ABB RobotStudio station: TPL01.rspag

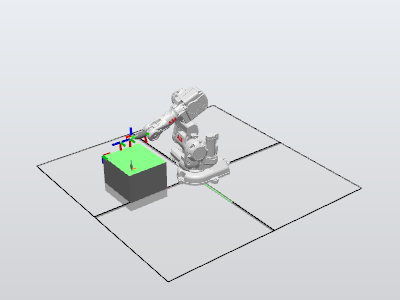
--- station ---
Station Project2 (saved by RobotStudio 25.5.11605.0)
Controller IRB140_6_81
  mechanical unit ROB_1: IRB140_6_81_C_03, 6 joints, base frame (0, 0, 0) mm
Layout (positions relative to the parent item):
  - IRB140_6_81_C_03 [mechanism, from %ABB.RobotStudio.Models.IRB140%\IRB140_6_81_C_G_03.rslib] at (0, 0, 0) mm; joint values [-0.1496, -0.0274, 0.4762, 2.8072, 0.4714, -2.4487] (rad or m)
  - Mesa [part], size 365 x 405 x 340 mm
  - Perno [part] at (730, 340, 177) mm, rotated rx 90 ry 0 rz -90 deg, size 20 x 100 x 20 mm
  - Pinza [mechanism] at (463, -60, 547) mm, rotated rx 90 ry 67.5 rz 90 deg
      TCP Pinza at (0, 0, 137) mm, rotated rx 0 ry 0 rz -22.5 deg
      links: Dummy
Attachment: Pinza is attached to IRB140_6_81_C_03 / Link6
Attachment: REF_Mesa is attached to Mesa
Attachment: REF_perno is attached to Perno
EventTableEntry 2314: ActivationMode=2, Cyclic=false, Group=, Trigger=DO_Pinza 2315, Actions=[EventTableActionAttach 2316], Comment=
EventTableTriggerIO 2315: Operator=0, IOValue=[1], IRC5Controller=? -1, SignalSource=IRB140_6_81 1261
EventTableActionAttach 2316: MountObject=false, FlangeIndext=0, FindNearest=false, AttachmentParent=Pinza 2308, AttachmentChild=Perno 2304, Offset=[X=1, Y=0, Z=0, W=0, X=0, Y=1, Z=0, W=0, X=0, Y=0, Z=1, W=0, X=0, Y=0, Z=0, W=1]
EventTableEntry 2317: ActivationMode=2, Cyclic=false, Group=, Trigger=DO_Pinza 2318, Actions=[EventTableActionDetach 2319], Comment=
EventTableTriggerIO 2318: Operator=0, IOValue=[0], IRC5Controller=? -1, SignalSource=IRB140_6_81 1261
EventTableActionDetach 2319: AttachmentParent=Pinza 2308, AttachmentChild=Perno 2304
Collision set CollisionSet_1: Perno against Mesa, near miss 0.005 m
EventTableTriggerIO 2517: Operator=0, IOValue=[1], IRC5Controller=? -1, SignalSource=IRB140_6_81 1261
EventTableTriggerIO 2518: Operator=0, IOValue=[0], IRC5Controller=? -1, SignalSource=IRB140_6_81 1261
Targets, tools, work objects and paths stored in the station and not in the controller backup, written as RAPID:
! task T_ROB1
MODULE Module1
  CONST robtarget home_10:=[[624.937,0,611],[1,0,0,0],[0,0,0,0],[9E+09,9E+09,9E+09,9E+09,9E+09,9E+09]];
ENDMODULE


--- Controller Data/IRB140_6_81/RAPID/TASK1/PROGMOD/CalibData.mod ---
MODULE CalibData
    PERS tooldata Pinza:=[TRUE,[[0,0,137],[0.98078528,0,0,-0.195090322]],[0.5,[0,0,100],[1,0,0,0],0,0,0]];
    TASK PERS wobjdata REF_Mesa:=[FALSE,TRUE,"",[[665,-400,260],[0,0,1,0]],[[0,0,0],[1,0,0,0]]];
    TASK PERS wobjdata REF_perno:=[FALSE,TRUE,"",[[400,180,130],[0.707106781,0.707106781,0,0]],[[0,0,0],[1,0,0,0]]];
ENDMODULE

--- Controller Data/IRB140_6_81/RAPID/TASK1/PROGMOD/Module1.mod ---
MODULE Module1
    CONST robtarget INSERTAR_PIEZA:=[[65,340,3],[1,0,0,0],[-1,1,-2,0],[9E+09,9E+09,9E+09,9E+09,9E+09,9E+09]];

    VAR robtarget TOMAR_PIEZA;
    !caso 1
    CONST robtarget TOMAR_PIEZA_VERTICAL:=[[0,0,10],[0.5,0.5,-0.5,0.5],[0,0,0,0],[9E+09,9E+09,9E+09,9E+09,9E+09,9E+09]];
    !caso 2
    CONST robtarget TOMAR_PIEZA_HORIZONTAL:=[[0,0,10],[1,0,0,0],[0,0,0,0],[9E+09,9E+09,9E+09,9E+09,9E+09,9E+09]];

    !Definicion de herramienta con perno
    PERS tooldata TCP_perno := [TRUE,[[83.1492,-34.4415,137],[0.69352,0.13795,0.69352,-0.13795]],[0.5,[0,0,100],[1,0,0,0],0,0,0]];

    !Transformacion pinza a perno
    VAR pose pinza_to_perno := [[90,0,0], [0,0,0,0]];

    VAR num MODO_PICK := 0; ! MODO_VERICAL = 0, MODO_HORIZONTAL = 1

    PROC main()

        init;
        test_path;

    ENDPROC

    PROC test_path()

        aproximar_perno;

        cerrar_pinza;

        aproximar_hueco;

        abrir_pinza;

        ir_inicio;

    ENDPROC


    PROC init()
        !Calculo de transformaciones de herramientas
        IF MODO_PICK = 0 THEN
            pinza_to_perno := [[90,0,0], OrientZYX(0,90,0)];
            TOMAR_PIEZA := TOMAR_PIEZA_VERTICAL;
        ELSE
            pinza_to_perno := [[0,0,90], OrientZYX(0,0,0)];
            TOMAR_PIEZA := TOMAR_PIEZA_HORIZONTAL;
        ENDIF

        TCP_perno.tframe := PoseMult(Pinza.tframe, pinza_to_perno);

        !Iniciar señales
        SetDO DO_Pinza,0;

    ENDPROC


    PROC aproximar_perno()
        VAR num offset:=50;

        !Aproximacion para agarrar
        MoveJ Offs(TOMAR_PIEZA,0,offset,0),v500,fine,Pinza\WObj:=REF_Perno;
        MoveL TOMAR_PIEZA,v1000,fine,Pinza\WObj:=REF_Perno;

    ENDPROC

    PROC cerrar_pinza()
        !Agarrar Pieza
        SetDO DO_Pinza,1;
    ENDPROC

    PROC aproximar_hueco()

        VAR num offset:=150;

        !Separase del punto de toma
        MoveL Offs(TOMAR_PIEZA,0,offset,0),v500,fine,Pinza\WObj:=REF_Perno;

        !Ir hasta el hueco
        MoveJ Offs(INSERTAR_PIEZA,0,0, -offset),v500,fine,TCP_perno\WObj:=REF_Mesa;

        !Insertar
        MoveL INSERTAR_PIEZA,v500,fine,TCP_perno\WObj:=REF_Mesa;

    ENDPROC


    PROC abrir_pinza()
        !Soltar Pieza
        SetDO DO_Pinza,0;
    ENDPROC

    PROC ir_inicio()

        VAR num offset:=200;

        !Salir del hueco
        MoveL Offs(INSERTAR_PIEZA,0,0, -offset),v500,fine,TCP_perno\WObj:=REF_Mesa;

        !Volver al inicio


    ENDPROC

ENDMODULE

--- Controller Data/IRB140_6_81/RAPID/TASK1/SYSMOD/LINKEDM.sys ---
%%%
  VERSION:1
  LANGUAGE:ENGLISH
%%%

MODULE LINKEDM (SYSMODULE)

! FOLLOWER
!     Name of electronically linked follower axis used by operator at teach pendent.
      PERS string l_f_axis_name{5}       :=  ["",  "", "", "", ""];

!     Name of the mechanical unit for follower axis.
      PERS string l_f_mecunt_n{5}  :=  ["", "", "", "", ""];

!     Linked follower axis number in the mechanical unit (first axis in mech. unit is number 1).
      PERS num l_f_axis_no{5}      :=  [0,          0,   0,  0,  0];

! MASTER
!     Name of the mechanical unit for linked master axis.
      PERS string l_m_mecunt_n{5} :=  ["", "", "", "", ""];

!     Linked master axis number in the mechanical unit (first axis in mech. unit is number 1).
!     See axis number table in documentation for different master mechanical units.
      PERS num l_m_axis_no{5}     :=  [0,  0,  0,  0,  0];

! POSITION OFFSET
!     The increase of the allowed offset position between the master and follower
!     positions, used when starting AUTO mode. As soon as the offset is decreased
!     the old configurated parameter is used.
!     Example: 3 => the configurated value of allowed offset is increased 3 times.
      PERS num offset_ratio{5}       :=  [10,  10,   10,  10,  10];

! SPEED RATIO
!     Speed_ratio used in AUTO and JOG modes [ very_slow   slow    normal    fast]
!     Value 1 = max allowed manual speed.
      CONST num speed_ratio {20}      := [0.01, 0.01, 0.01, 0.01, 0.01,
                                          0.05, 0.05, 0.05, 0.05, 0.05,
                                          0.20, 0.20, 0.20, 0.20, 0.20,
                                          1.00, 1.00, 1.00, 1.00, 1.00];

! STEP SIZE
!     Displacement position used in JOG mode for each activation of positive or
!     negative movement.                  [very_short    short   normal   long]
!     Unit degees or meter.
      CONST num displacement {20}     := [0.001, 0.001, 0.001, 0.001, 0.001,
                                          0.005, 0.005, 0.005, 0.005, 0.005,
                                          0.020, 0.020, 0.020, 0.020, 0.020,
                                          0.100, 0.100, 0.100, 0.100, 0.100];


!-------------------------------------------------------------
 PROC Linked_m ()
      Linked_m_exe ;
 ENDPROC
ENDMODULE

--- Controller Data/IRB140_6_81/SYSPAR/EIO.cfg ---
EIO:CFG_1.0:6:1::
#
EIO_SIGNAL:

      -Name "DO_Pinza" -SignalType "DO" -Access "All"
